FUNCTION_BLOCK FB_Simu_NT
VAR_INPUT

END_VAR

VAR_OUTPUT
	iOUT_TC_Water_1			: INT;
	iOUT_TC_Water_2			: INT;
	iOUT_CJC_Value			: INT;
	iOUT_ToolID_Value		: INT;
	bOUT_WaterFlow_1		: BOOL;
	bOUT_WaterFlow_2		: BOOL;
	bOUT_AirPressure		: BOOL;
	bOUT_TC_Water_1_Error	: BOOL;
	bOUT_TC_Water_2_Error	: BOOL;
	bOUT_CJC_Error			: BOOL;
	bOUT_ToolID_Error		: INT;
END_VAR
VAR
END_VAR

// NETWORK 1

END_FUNCTION_BLOCK

(* stored: Version 1.1.0.1, ProductVersion 3.1.4024.12
   POU FB_Simu_NT: Id {9ea71bbd-eae6-4317-8eaf-7d51dd590fd6}, SpecialFunc None *)
